(* Logix 5000 project; controller L3 vendor 1 type 14 code 92 rev 20.12; software revision 20.04; part 3 of 9 *)
(* tags used below, declared in another part *)
   B3 : DINT[100];
   N20 : DINT[200];
   N21 : DINT[200];
   N7 : DINT[200];
   N9 : DINT[200];   // niveau decapage vers lancy (n9[10) ;;N9[70]
   S_SP_DEC : DINT;
   T4 : TIMER[180];
(* _2_GENERAL, continued *)

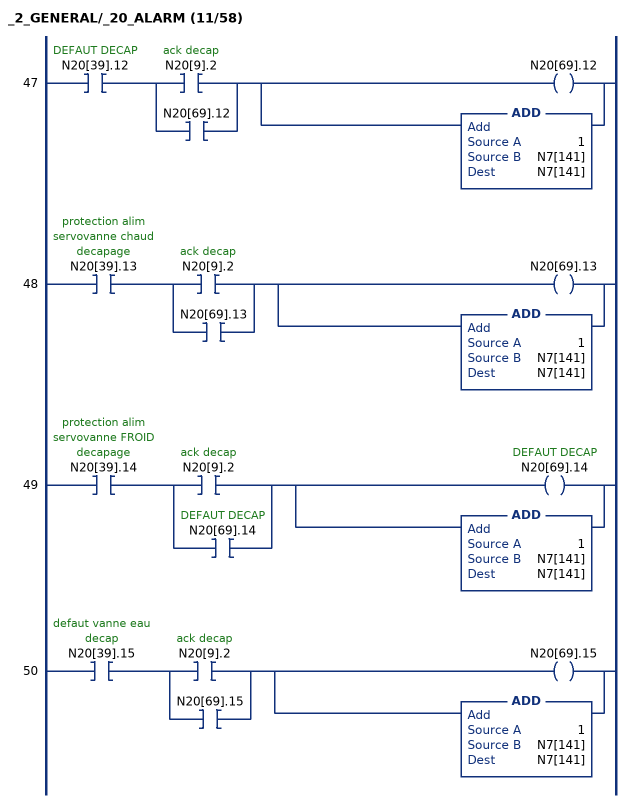
   [picture p26: _2_GENERAL/_20_ALARM rungs 47-50]
   47: XIC(N20[39].12)[XIC(N20[9].2) ,XIC(N20[69].12) ][OTE(N20[69].12) ,ADD(1,N7[141],N7[141]) ];
   48: XIC(N20[39].13)[XIC(N20[9].2) ,XIC(N20[69].13) ][OTE(N20[69].13) ,ADD(1,N7[141],N7[141]) ];
   49: XIC(N20[39].14)[XIC(N20[9].2) ,XIC(N20[69].14) ][OTE(N20[69].14) ,ADD(1,N7[141],N7[141]) ];
   50: XIC(N20[39].15)[XIC(N20[9].2) ,XIC(N20[69].15) ][OTE(N20[69].15) ,ADD(1,N7[141],N7[141]) ];
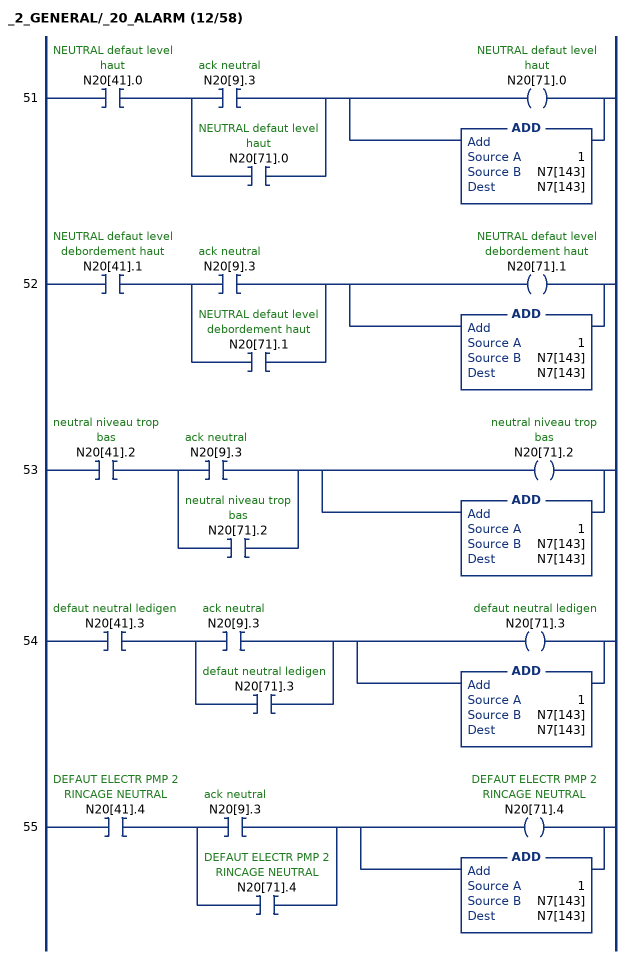
   51: XIC(N20[41].0)[XIC(N20[9].3) ,XIC(N20[71].0) ][OTE(N20[71].0) ,ADD(1,N7[143],N7[143]) ];
   52: XIC(N20[41].1)[XIC(N20[9].3) ,XIC(N20[71].1) ][OTE(N20[71].1) ,ADD(1,N7[143],N7[143]) ];
   53: XIC(N20[41].2)[XIC(N20[9].3) ,XIC(N20[71].2) ][OTE(N20[71].2) ,ADD(1,N7[143],N7[143]) ];
   54: XIC(N20[41].3)[XIC(N20[9].3) ,XIC(N20[71].3) ][OTE(N20[71].3) ,ADD(1,N7[143],N7[143]) ];
   55: XIC(N20[41].4)[XIC(N20[9].3) ,XIC(N20[71].4) ][OTE(N20[71].4) ,ADD(1,N7[143],N7[143]) ];
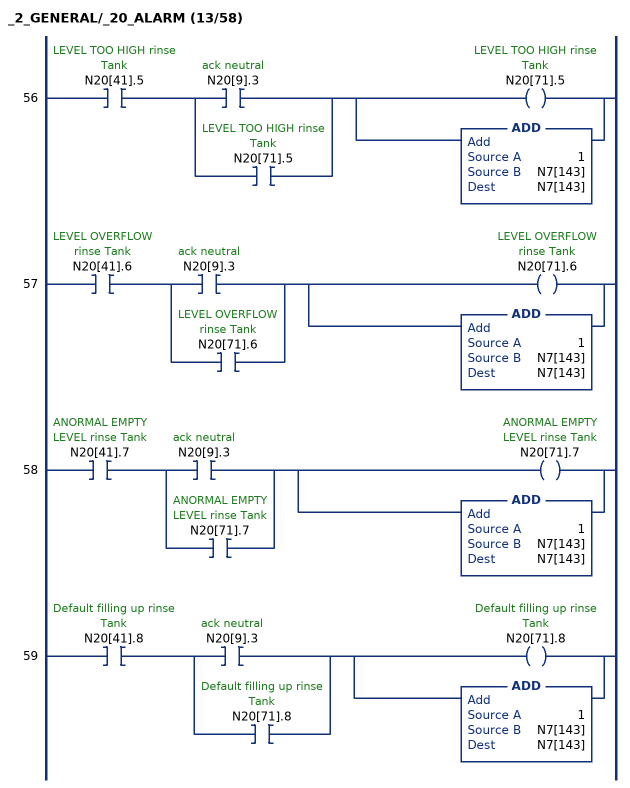
   56: XIC(N20[41].5)[XIC(N20[9].3) ,XIC(N20[71].5) ][OTE(N20[71].5) ,ADD(1,N7[143],N7[143]) ];
   57: XIC(N20[41].6)[XIC(N20[9].3) ,XIC(N20[71].6) ][OTE(N20[71].6) ,ADD(1,N7[143],N7[143]) ];
   58: XIC(N20[41].7)[XIC(N20[9].3) ,XIC(N20[71].7) ][OTE(N20[71].7) ,ADD(1,N7[143],N7[143]) ];
   59: XIC(N20[41].8)[XIC(N20[9].3) ,XIC(N20[71].8) ][OTE(N20[71].8) ,ADD(1,N7[143],N7[143]) ];
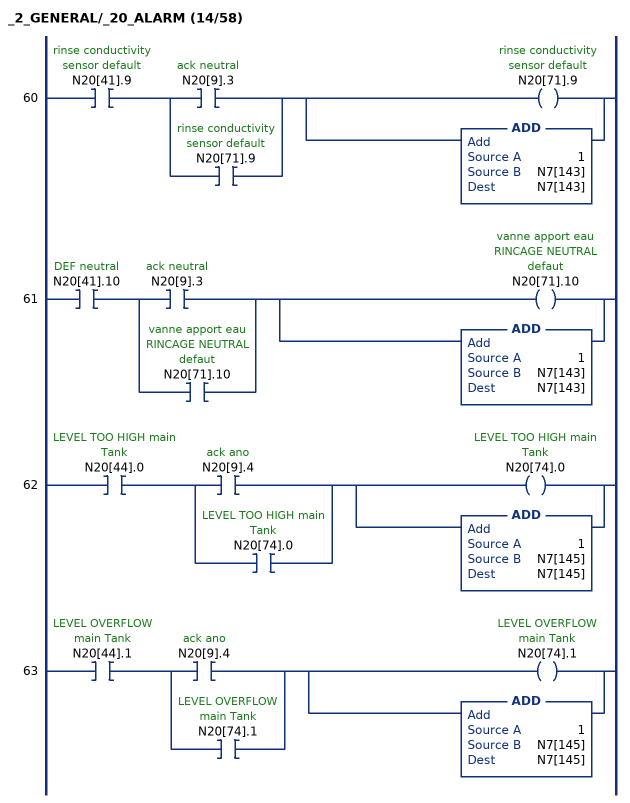
   60: XIC(N20[41].9)[XIC(N20[9].3) ,XIC(N20[71].9) ][OTE(N20[71].9) ,ADD(1,N7[143],N7[143]) ];
   61: XIC(N20[41].10)[XIC(N20[9].3) ,XIC(N20[71].10) ][OTE(N20[71].10) ,ADD(1,N7[143],N7[143]) ];
   62: XIC(N20[44].0)[XIC(N20[9].4) ,XIC(N20[74].0) ][OTE(N20[74].0) ,ADD(1,N7[145],N7[145]) ];
   63: XIC(N20[44].1)[XIC(N20[9].4) ,XIC(N20[74].1) ][OTE(N20[74].1) ,ADD(1,N7[145],N7[145]) ];
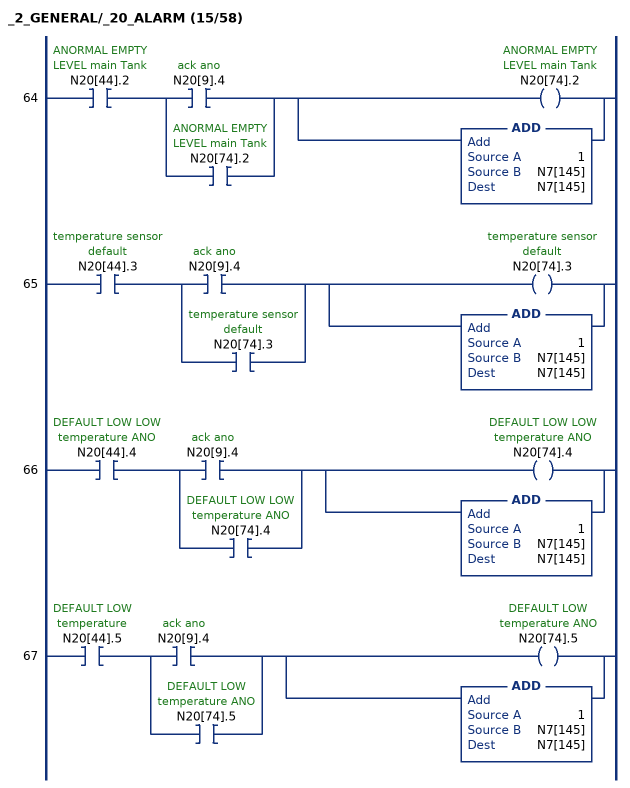
   64: XIC(N20[44].2)[XIC(N20[9].4) ,XIC(N20[74].2) ][OTE(N20[74].2) ,ADD(1,N7[145],N7[145]) ];
   65: XIC(N20[44].3)[XIC(N20[9].4) ,XIC(N20[74].3) ][OTE(N20[74].3) ,ADD(1,N7[145],N7[145]) ];
   66: XIC(N20[44].4)[XIC(N20[9].4) ,XIC(N20[74].4) ][OTE(N20[74].4) ,ADD(1,N7[145],N7[145]) ];
   67: XIC(N20[44].5)[XIC(N20[9].4) ,XIC(N20[74].5) ][OTE(N20[74].5) ,ADD(1,N7[145],N7[145]) ];
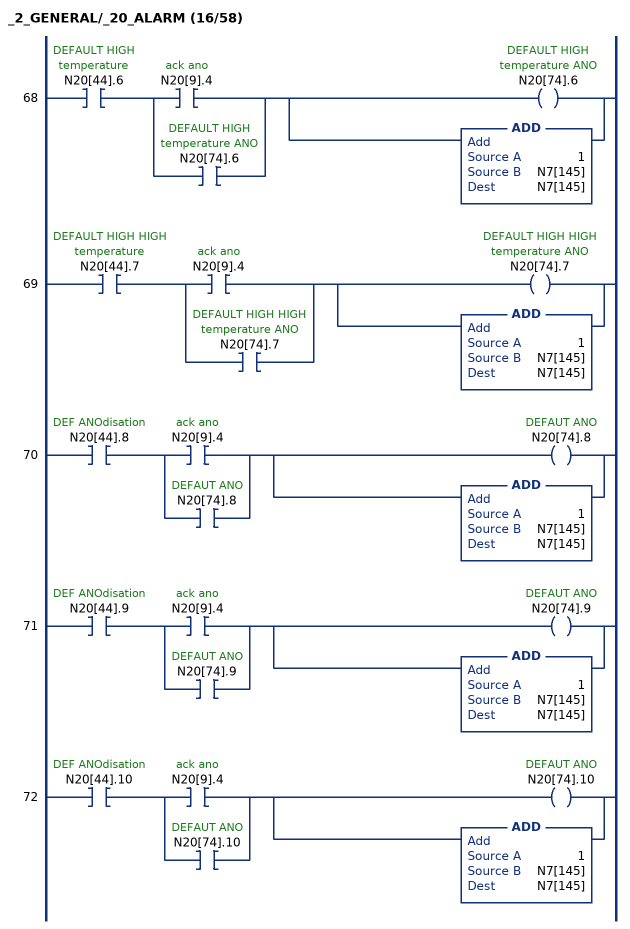
   68: XIC(N20[44].6)[XIC(N20[9].4) ,XIC(N20[74].6) ][OTE(N20[74].6) ,ADD(1,N7[145],N7[145]) ];
   69: XIC(N20[44].7)[XIC(N20[9].4) ,XIC(N20[74].7) ][OTE(N20[74].7) ,ADD(1,N7[145],N7[145]) ];
   70: XIC(N20[44].8)[XIC(N20[9].4) ,XIC(N20[74].8) ][OTE(N20[74].8) ,ADD(1,N7[145],N7[145]) ];
   71: XIC(N20[44].9)[XIC(N20[9].4) ,XIC(N20[74].9) ][OTE(N20[74].9) ,ADD(1,N7[145],N7[145]) ];
   72: XIC(N20[44].10)[XIC(N20[9].4) ,XIC(N20[74].10) ][OTE(N20[74].10) ,ADD(1,N7[145],N7[145]) ];
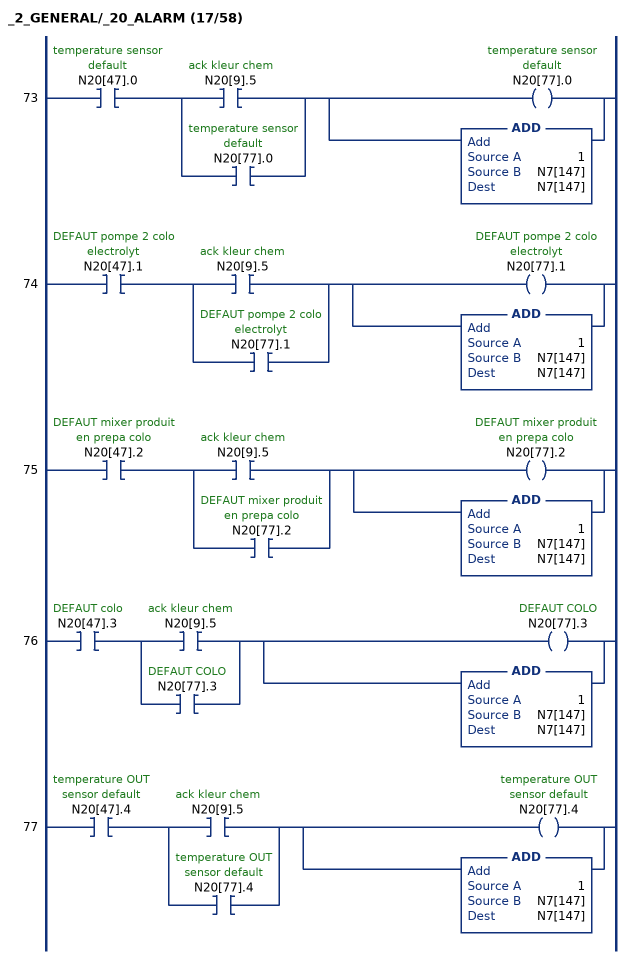
   73: XIC(N20[47].0)[XIC(N20[9].5) ,XIC(N20[77].0) ][OTE(N20[77].0) ,ADD(1,N7[147],N7[147]) ];
   74: XIC(N20[47].1)[XIC(N20[9].5) ,XIC(N20[77].1) ][OTE(N20[77].1) ,ADD(1,N7[147],N7[147]) ];
   75: XIC(N20[47].2)[XIC(N20[9].5) ,XIC(N20[77].2) ][OTE(N20[77].2) ,ADD(1,N7[147],N7[147]) ];
   76: XIC(N20[47].3)[XIC(N20[9].5) ,XIC(N20[77].3) ][OTE(N20[77].3) ,ADD(1,N7[147],N7[147]) ];
   77: XIC(N20[47].4)[XIC(N20[9].5) ,XIC(N20[77].4) ][OTE(N20[77].4) ,ADD(1,N7[147],N7[147]) ];
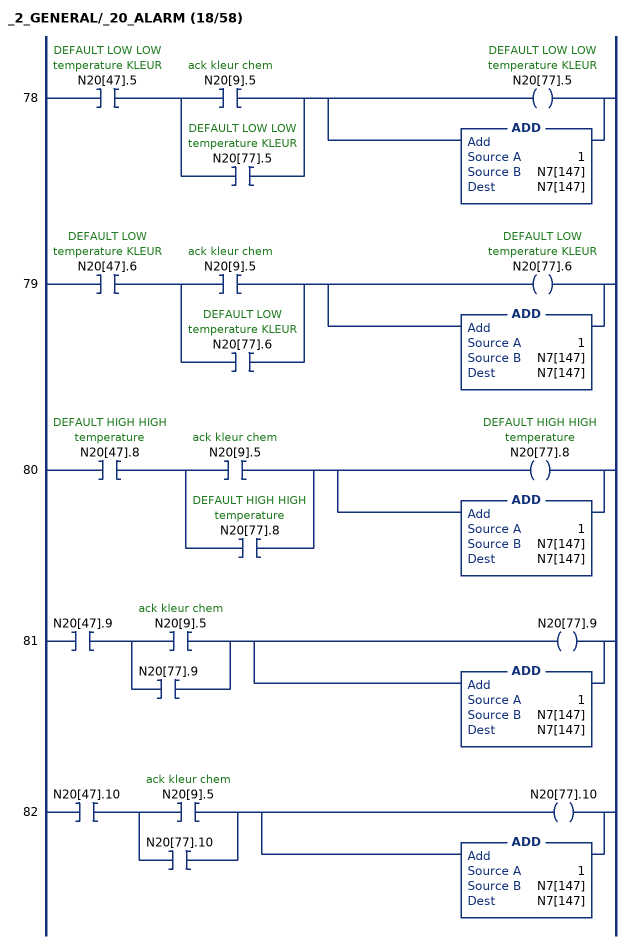
   78: XIC(N20[47].5)[XIC(N20[9].5) ,XIC(N20[77].5) ][OTE(N20[77].5) ,ADD(1,N7[147],N7[147]) ];
   79: XIC(N20[47].6)[XIC(N20[9].5) ,XIC(N20[77].6) ][OTE(N20[77].6) ,ADD(1,N7[147],N7[147]) ];
   80: XIC(N20[47].8)[XIC(N20[9].5) ,XIC(N20[77].8) ][OTE(N20[77].8) ,ADD(1,N7[147],N7[147]) ];
   81: XIC(N20[47].9)[XIC(N20[9].5) ,XIC(N20[77].9) ][OTE(N20[77].9) ,ADD(1,N7[147],N7[147]) ];
   82: XIC(N20[47].10)[XIC(N20[9].5) ,XIC(N20[77].10) ][OTE(N20[77].10) ,ADD(1,N7[147],N7[147]) ];
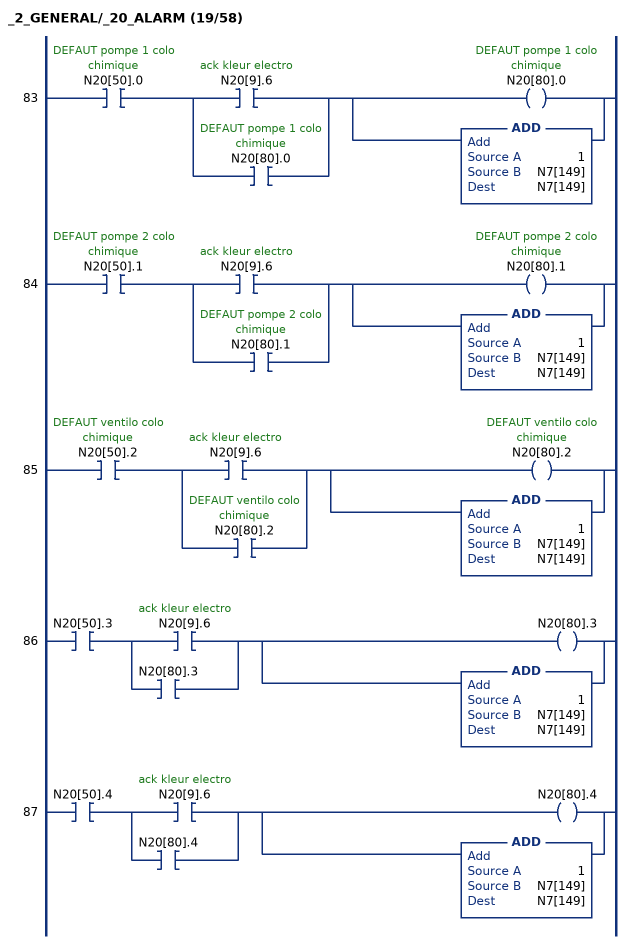
   83: XIC(N20[50].0)[XIC(N20[9].6) ,XIC(N20[80].0) ][OTE(N20[80].0) ,ADD(1,N7[149],N7[149]) ];
   84: XIC(N20[50].1)[XIC(N20[9].6) ,XIC(N20[80].1) ][OTE(N20[80].1) ,ADD(1,N7[149],N7[149]) ];
   85: XIC(N20[50].2)[XIC(N20[9].6) ,XIC(N20[80].2) ][OTE(N20[80].2) ,ADD(1,N7[149],N7[149]) ];
   86: XIC(N20[50].3)[XIC(N20[9].6) ,XIC(N20[80].3) ][OTE(N20[80].3) ,ADD(1,N7[149],N7[149]) ];
   87: XIC(N20[50].4)[XIC(N20[9].6) ,XIC(N20[80].4) ][OTE(N20[80].4) ,ADD(1,N7[149],N7[149]) ];
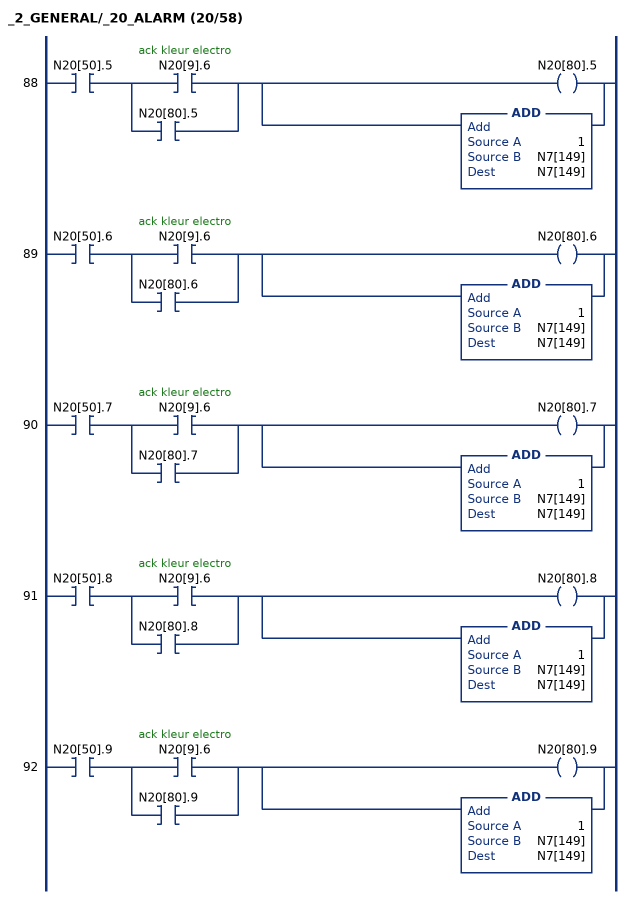
   88: XIC(N20[50].5)[XIC(N20[9].6) ,XIC(N20[80].5) ][OTE(N20[80].5) ,ADD(1,N7[149],N7[149]) ];
   89: XIC(N20[50].6)[XIC(N20[9].6) ,XIC(N20[80].6) ][OTE(N20[80].6) ,ADD(1,N7[149],N7[149]) ];
   90: XIC(N20[50].7)[XIC(N20[9].6) ,XIC(N20[80].7) ][OTE(N20[80].7) ,ADD(1,N7[149],N7[149]) ];
   91: XIC(N20[50].8)[XIC(N20[9].6) ,XIC(N20[80].8) ][OTE(N20[80].8) ,ADD(1,N7[149],N7[149]) ];
   92: XIC(N20[50].9)[XIC(N20[9].6) ,XIC(N20[80].9) ][OTE(N20[80].9) ,ADD(1,N7[149],N7[149]) ];
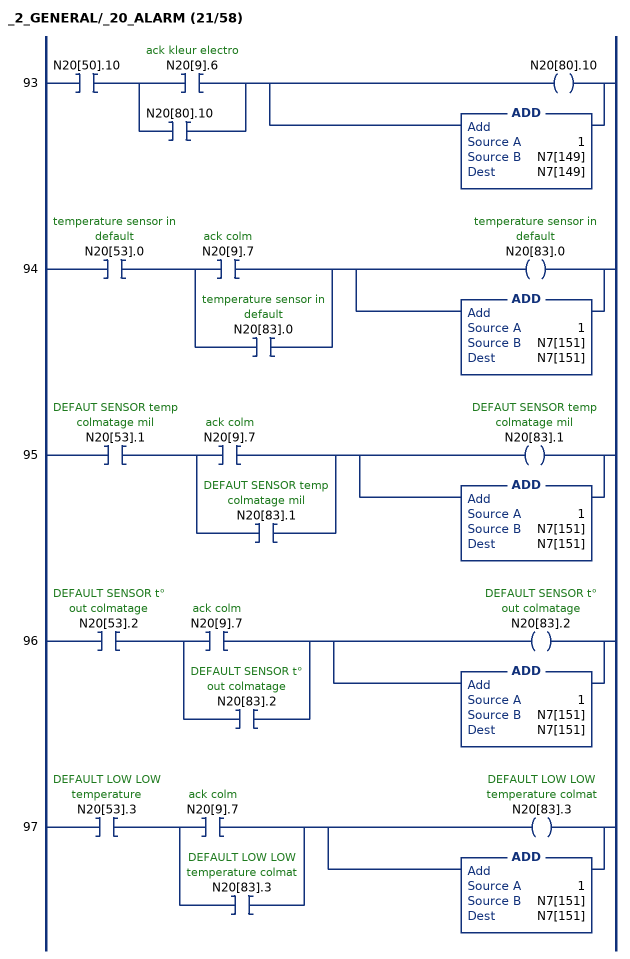
   93: XIC(N20[50].10)[XIC(N20[9].6) ,XIC(N20[80].10) ][OTE(N20[80].10) ,ADD(1,N7[149],N7[149]) ];
   94: XIC(N20[53].0)[XIC(N20[9].7) ,XIC(N20[83].0) ][OTE(N20[83].0) ,ADD(1,N7[151],N7[151]) ];
   95: XIC(N20[53].1)[XIC(N20[9].7) ,XIC(N20[83].1) ][OTE(N20[83].1) ,ADD(1,N7[151],N7[151]) ];
   96: XIC(N20[53].2)[XIC(N20[9].7) ,XIC(N20[83].2) ][OTE(N20[83].2) ,ADD(1,N7[151],N7[151]) ];
   97: XIC(N20[53].3)[XIC(N20[9].7) ,XIC(N20[83].3) ][OTE(N20[83].3) ,ADD(1,N7[151],N7[151]) ];
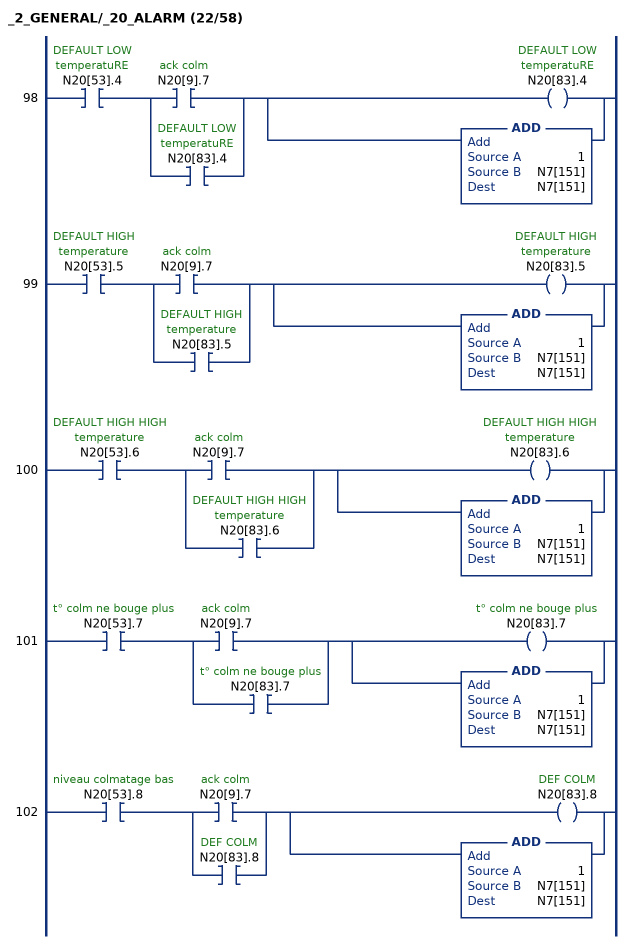
   98: XIC(N20[53].4)[XIC(N20[9].7) ,XIC(N20[83].4) ][OTE(N20[83].4) ,ADD(1,N7[151],N7[151]) ];
   99: XIC(N20[53].5)[XIC(N20[9].7) ,XIC(N20[83].5) ][OTE(N20[83].5) ,ADD(1,N7[151],N7[151]) ];
   100: XIC(N20[53].6)[XIC(N20[9].7) ,XIC(N20[83].6) ][OTE(N20[83].6) ,ADD(1,N7[151],N7[151]) ];
   101: XIC(N20[53].7)[XIC(N20[9].7) ,XIC(N20[83].7) ][OTE(N20[83].7) ,ADD(1,N7[151],N7[151]) ];
   102: XIC(N20[53].8)[XIC(N20[9].7) ,XIC(N20[83].8) ][OTE(N20[83].8) ,ADD(1,N7[151],N7[151]) ];
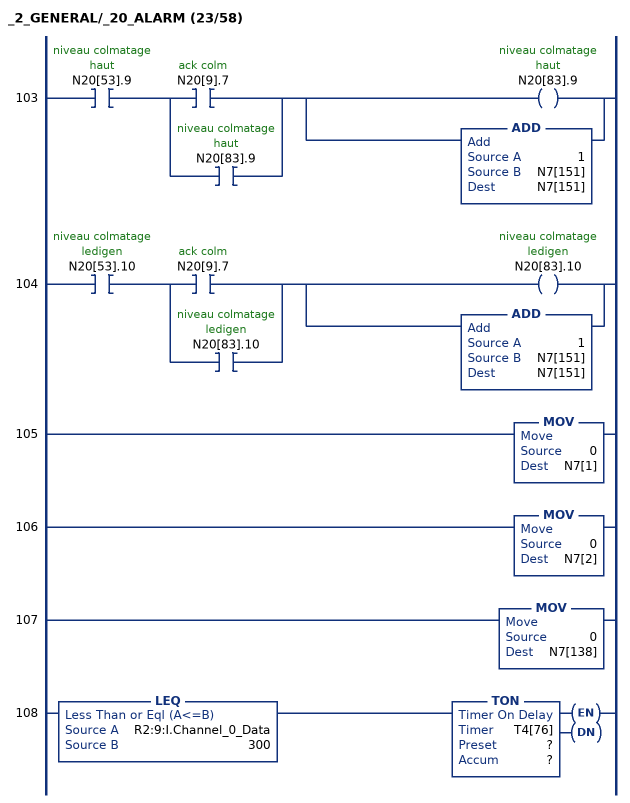
   103: XIC(N20[53].9)[XIC(N20[9].7) ,XIC(N20[83].9) ][OTE(N20[83].9) ,ADD(1,N7[151],N7[151]) ];
   104: XIC(N20[53].10)[XIC(N20[9].7) ,XIC(N20[83].10) ][OTE(N20[83].10) ,ADD(1,N7[151],N7[151]) ];
   105: MOV(0,N7[1]);
   106: MOV(0,N7[2]);
   107: MOV(0,N7[138]);
   108: LEQ(R2:9:I.Channel_0_Data,300)TON(T4[76],?,?);
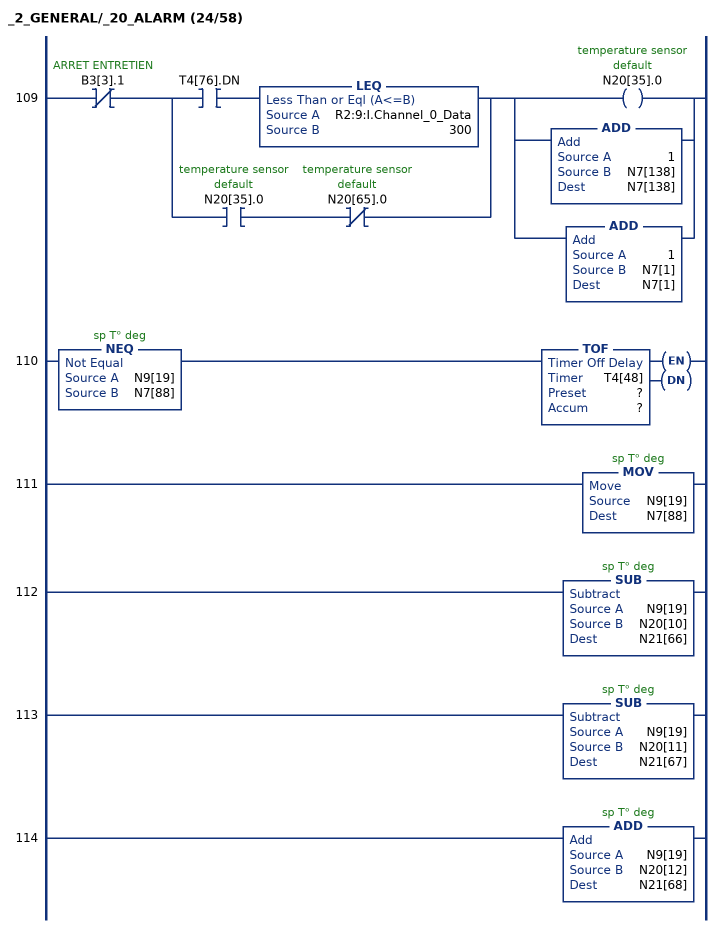
   109: XIO(B3[3].1)[XIC(T4[76].DN) LEQ(R2:9:I.Channel_0_Data,300) ,XIC(N20[35].0) XIO(N20[65].0) ][OTE(N20[35].0) ,ADD(1,N7[138],N7[138]) ,ADD(1,N7[1],N7[1]) ];
   110: NEQ(N9[19],N7[88])TOF(T4[48],?,?);
   111: MOV(N9[19],N7[88]);
   112: SUB(N9[19],N20[10],N21[66]);
   113: SUB(N9[19],N20[11],N21[67]);
   114: ADD(N9[19],N20[12],N21[68]);
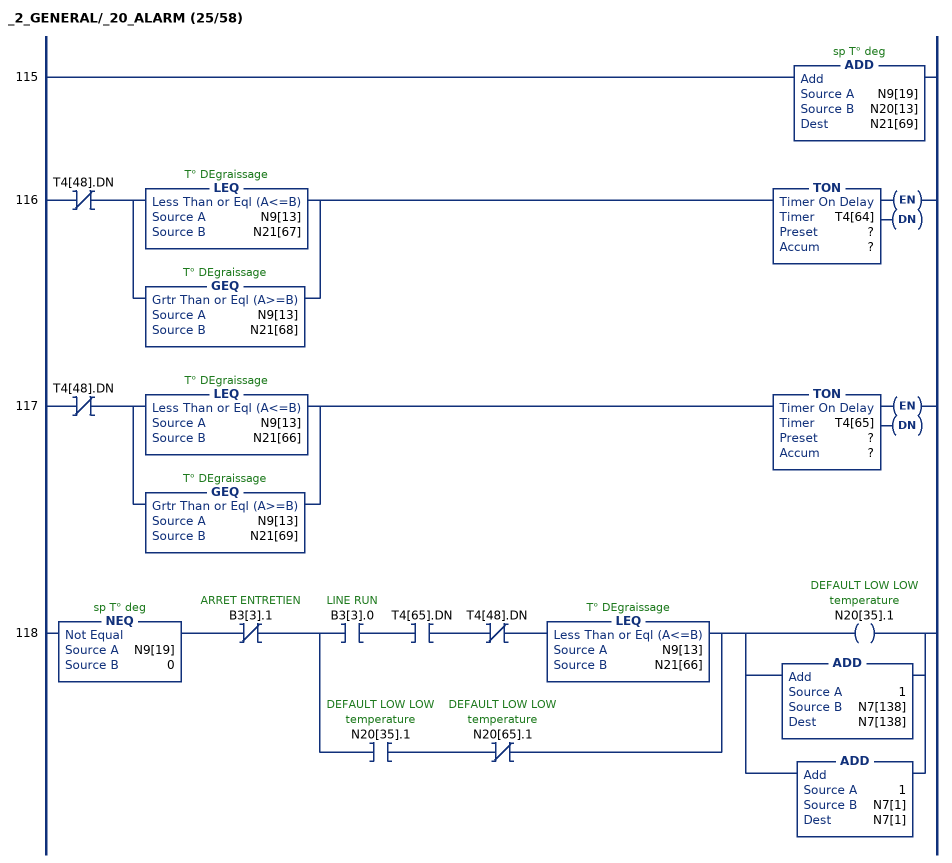
   115: ADD(N9[19],N20[13],N21[69]);
   116: XIO(T4[48].DN)[LEQ(N9[13],N21[67]) ,GEQ(N9[13],N21[68]) ]TON(T4[64],?,?);
   117: XIO(T4[48].DN)[LEQ(N9[13],N21[66]) ,GEQ(N9[13],N21[69]) ]TON(T4[65],?,?);
   118: NEQ(N9[19],0)XIO(B3[3].1)[XIC(B3[3].0) XIC(T4[65].DN) XIO(T4[48].DN) LEQ(N9[13],N21[66]) ,XIC(N20[35].1) XIO(N20[65].1) ][OTE(N20[35].1) ,ADD(1,N7[138],N7[138]) ,ADD(1,N7[1],N7[1]) ];
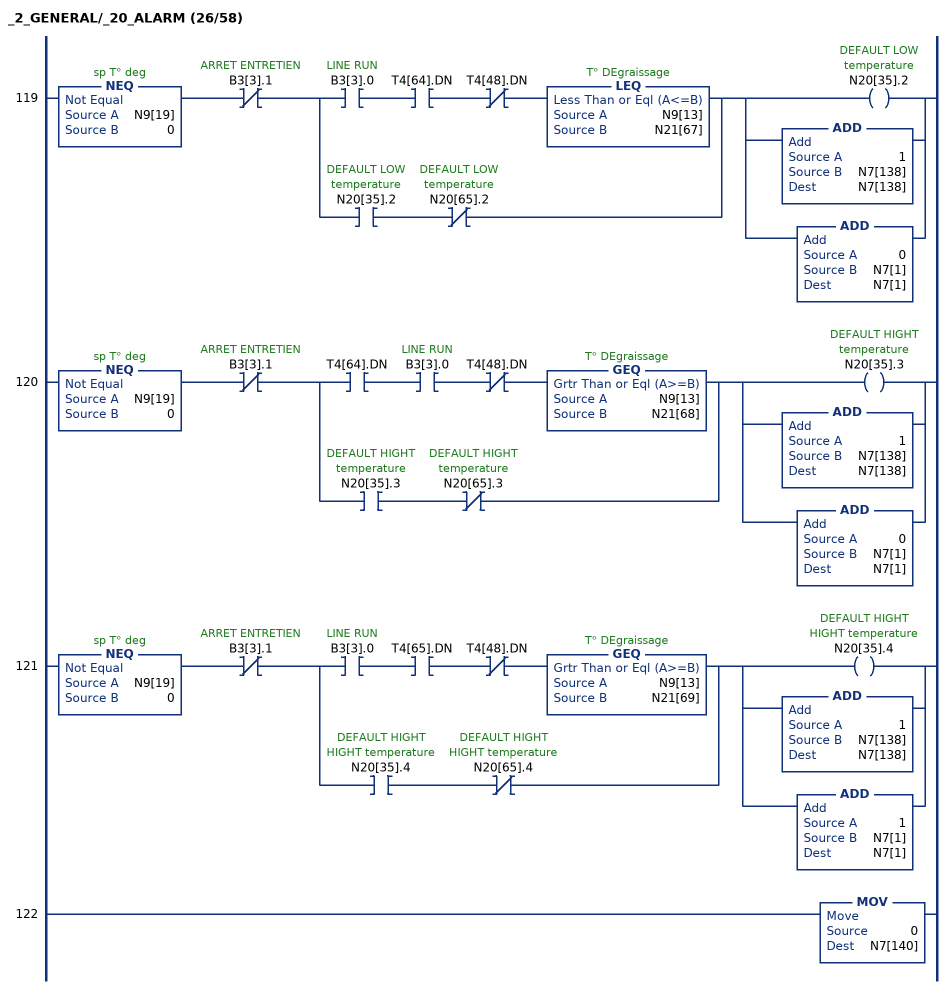
   119: NEQ(N9[19],0)XIO(B3[3].1)[XIC(B3[3].0) XIC(T4[64].DN) XIO(T4[48].DN) LEQ(N9[13],N21[67]) ,XIC(N20[35].2) XIO(N20[65].2) ][OTE(N20[35].2) ,ADD(1,N7[138],N7[138]) ,ADD(0,N7[1],N7[1]) ];
   120: NEQ(N9[19],0)XIO(B3[3].1)[XIC(T4[64].DN) XIC(B3[3].0) XIO(T4[48].DN) GEQ(N9[13],N21[68]) ,XIC(N20[35].3) XIO(N20[65].3) ][OTE(N20[35].3) ,ADD(1,N7[138],N7[138]) ,ADD(0,N7[1],N7[1]) ];
   121: NEQ(N9[19],0)XIO(B3[3].1)[XIC(B3[3].0) XIC(T4[65].DN) XIO(T4[48].DN) GEQ(N9[13],N21[69]) ,XIC(N20[35].4) XIO(N20[65].4) ][OTE(N20[35].4) ,ADD(1,N7[138],N7[138]) ,ADD(1,N7[1],N7[1]) ];
   122: MOV(0,N7[140]);
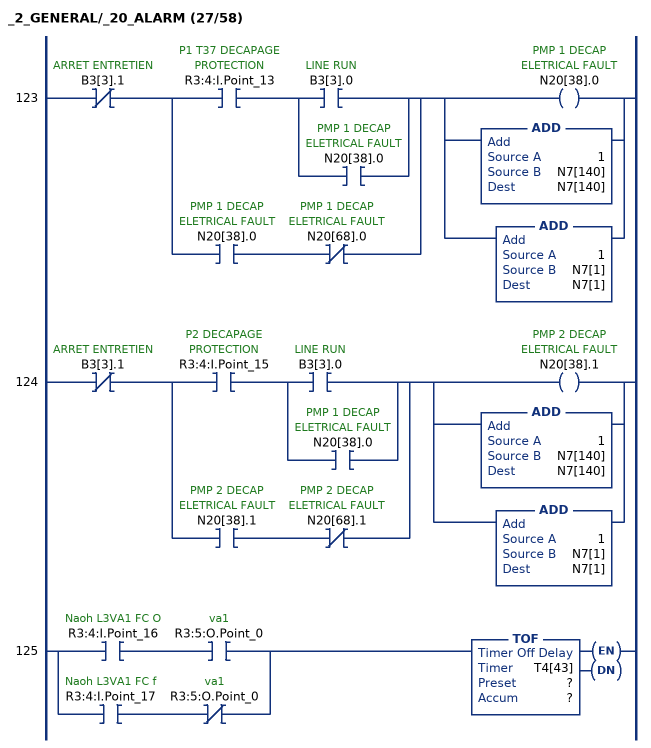
   123: XIO(B3[3].1)[XIC(R3:4:I.Point_13) [XIC(B3[3].0) ,XIC(N20[38].0) ] ,XIC(N20[38].0) XIO(N20[68].0) ][OTE(N20[38].0) ,ADD(1,N7[140],N7[140]) ,ADD(1,N7[1],N7[1]) ];
   124: XIO(B3[3].1)[XIC(R3:4:I.Point_15) [XIC(B3[3].0) ,XIC(N20[38].0) ] ,XIC(N20[38].1) XIO(N20[68].1) ][OTE(N20[38].1) ,ADD(1,N7[140],N7[140]) ,ADD(1,N7[1],N7[1]) ];
   125: [XIC(R3:4:I.Point_16) XIC(R3:5:O.Point_0) ,XIC(R3:4:I.Point_17) XIO(R3:5:O.Point_0) ]TOF(T4[43],?,?);
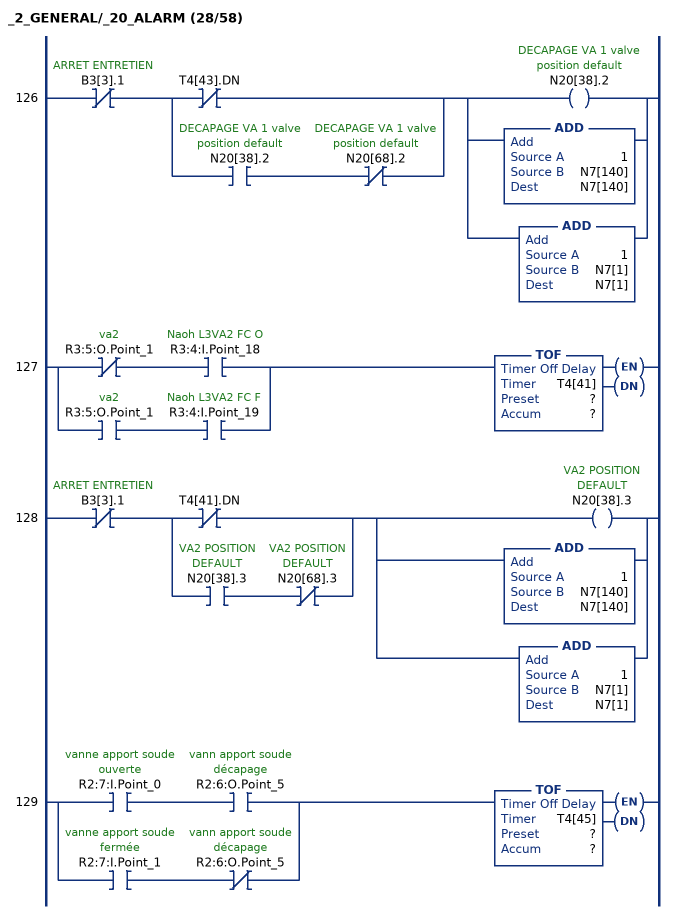
   126: XIO(B3[3].1)[XIO(T4[43].DN) ,XIC(N20[38].2) XIO(N20[68].2) ][OTE(N20[38].2) ,ADD(1,N7[140],N7[140]) ,ADD(1,N7[1],N7[1]) ];
   127: [XIO(R3:5:O.Point_1) XIC(R3:4:I.Point_18) ,XIC(R3:5:O.Point_1) XIC(R3:4:I.Point_19) ]TOF(T4[41],?,?);
   128: XIO(B3[3].1)[XIO(T4[41].DN) ,XIC(N20[38].3) XIO(N20[68].3) ][OTE(N20[38].3) ,ADD(1,N7[140],N7[140]) ,ADD(1,N7[1],N7[1]) ];
   129: [XIC(R2:7:I.Point_0) XIC(R2:6:O.Point_5) ,XIC(R2:7:I.Point_1) XIO(R2:6:O.Point_5) ]TOF(T4[45],?,?);
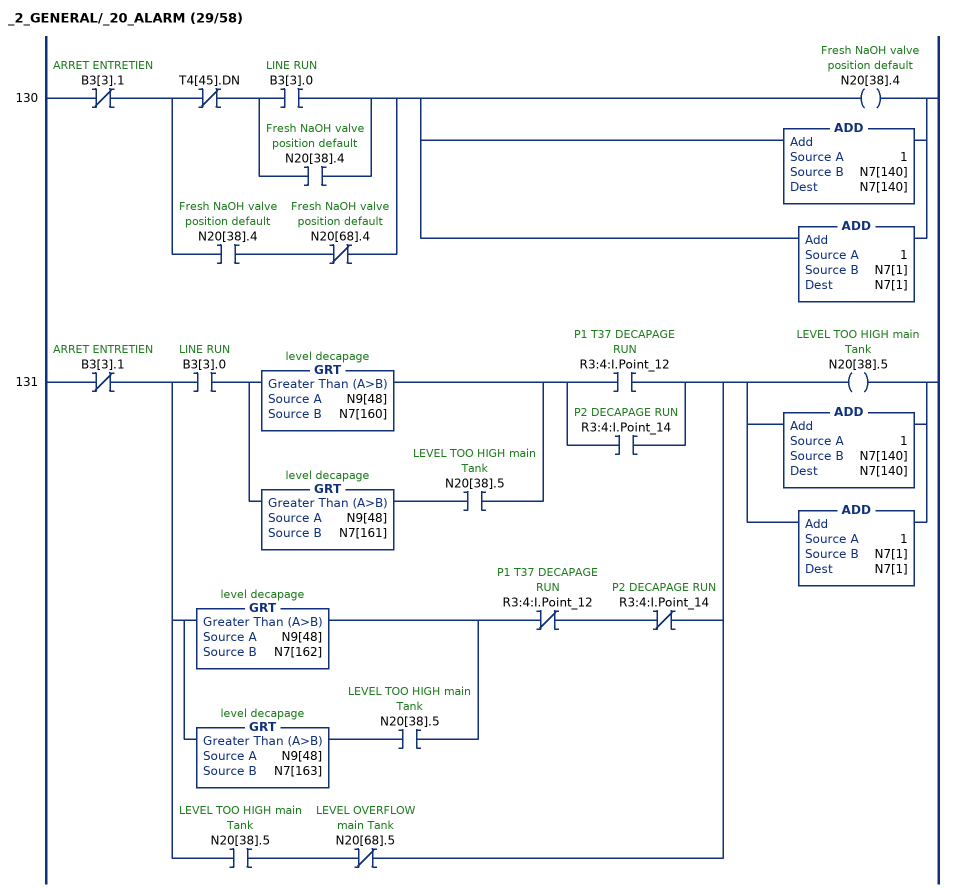
   130: XIO(B3[3].1)[XIO(T4[45].DN) [XIC(B3[3].0) ,XIC(N20[38].4) ] ,XIC(N20[38].4) XIO(N20[68].4) ][OTE(N20[38].4) ,ADD(1,N7[140],N7[140]) ,ADD(1,N7[1],N7[1]) ];
   131: XIO(B3[3].1)[XIC(B3[3].0) [GRT(N9[48],N7[160]) ,GRT(N9[48],N7[161]) XIC(N20[38].5) ] [XIC(R3:4:I.Point_12) ,XIC(R3:4:I.Point_14) ] ,[GRT(N9[48],N7[162]) ,GRT(N9[48],N7[163]) XIC(N20[38].5) ] XIO(R3:4:I.Point_12) XIO(R3:4:I.Point_14) ,XIC(N20[38].5) XIO(N20[68].5) ][OTE(N20[38].5) ,ADD(1,N7[140],N7[140]) ,ADD(1,N7[1],N7[1]) ];
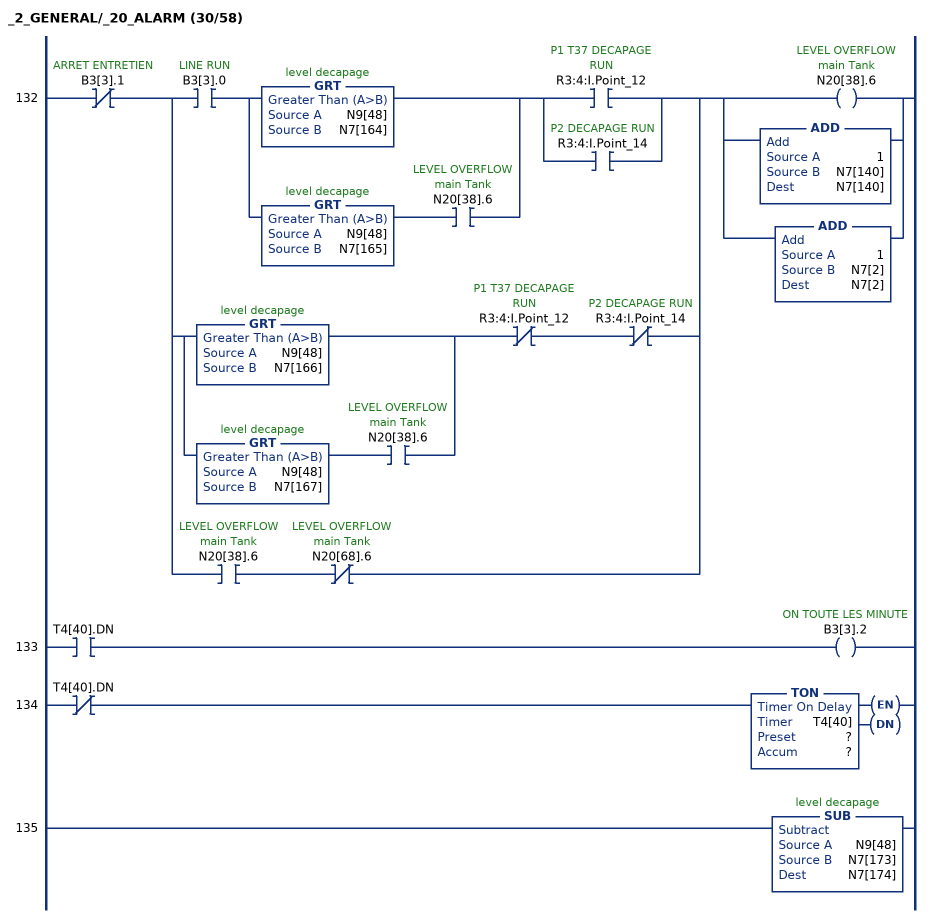
   132: XIO(B3[3].1)[XIC(B3[3].0) [GRT(N9[48],N7[164]) ,GRT(N9[48],N7[165]) XIC(N20[38].6) ] [XIC(R3:4:I.Point_12) ,XIC(R3:4:I.Point_14) ] ,[GRT(N9[48],N7[166]) ,GRT(N9[48],N7[167]) XIC(N20[38].6) ] XIO(R3:4:I.Point_12) XIO(R3:4:I.Point_14) ,XIC(N20[38].6) XIO(N20[68].6) ][OTE(N20[38].6) ,ADD(1,N7[140],N7[140]) ,ADD(1,N7[2],N7[2]) ];
   133: XIC(T4[40].DN)OTE(B3[3].2);
   134: XIO(T4[40].DN)TON(T4[40],?,?);
   135: SUB(N9[48],N7[173],N7[174]);
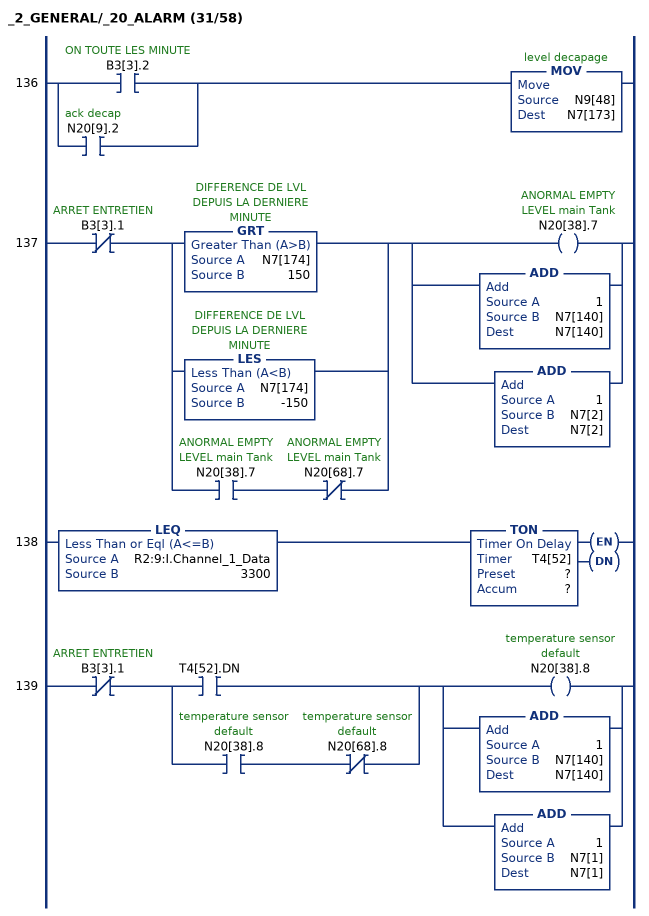
   136: [XIC(B3[3].2) ,XIC(N20[9].2) ]MOV(N9[48],N7[173]);
   137: XIO(B3[3].1)[GRT(N7[174],150) ,LES(N7[174],-150) ,XIC(N20[38].7) XIO(N20[68].7) ][OTE(N20[38].7) ,ADD(1,N7[140],N7[140]) ,ADD(1,N7[2],N7[2]) ];
   138: LEQ(R2:9:I.Channel_1_Data,3300)TON(T4[52],?,?);
   139: XIO(B3[3].1)[XIC(T4[52].DN) ,XIC(N20[38].8) XIO(N20[68].8) ][OTE(N20[38].8) ,ADD(1,N7[140],N7[140]) ,ADD(1,N7[1],N7[1]) ];
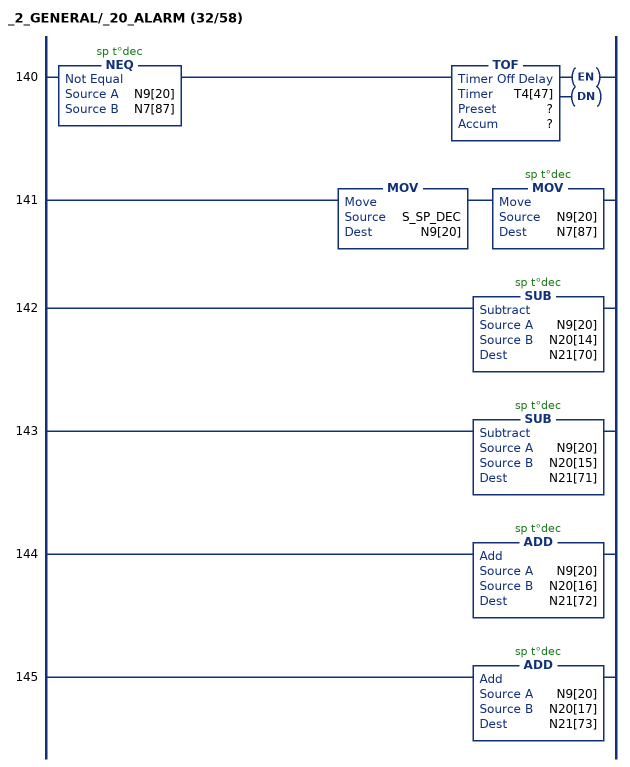
   140: NEQ(N9[20],N7[87])TOF(T4[47],?,?);
   141: MOV(S_SP_DEC,N9[20])MOV(N9[20],N7[87]);
   142: SUB(N9[20],N20[14],N21[70]);
   143: SUB(N9[20],N20[15],N21[71]);
   144: ADD(N9[20],N20[16],N21[72]);
   145: ADD(N9[20],N20[17],N21[73]);
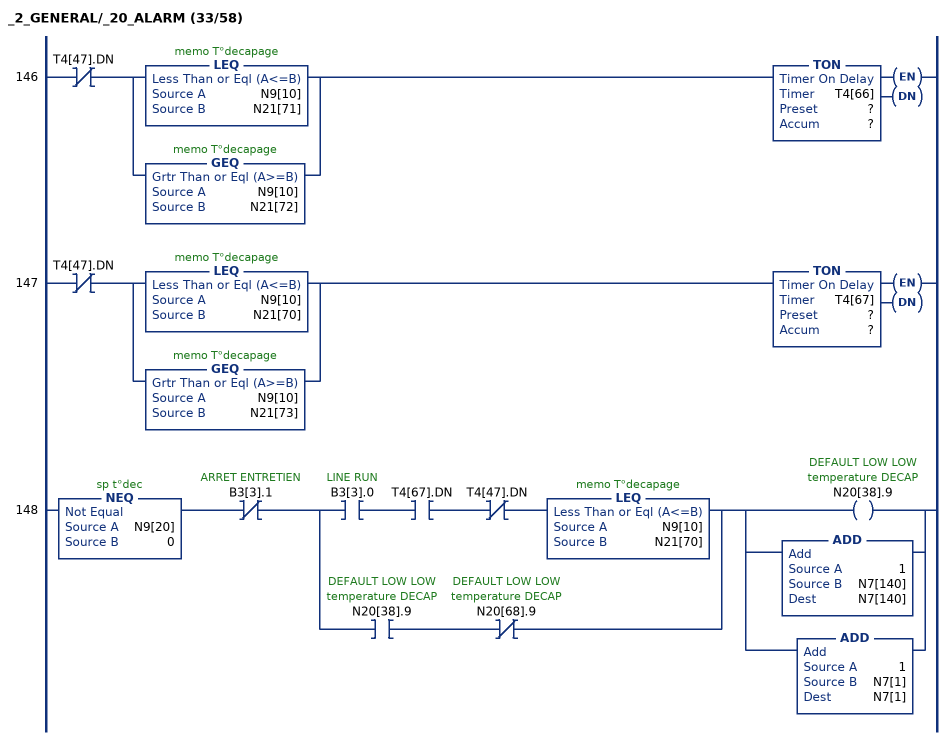
   146: XIO(T4[47].DN)[LEQ(N9[10],N21[71]) ,GEQ(N9[10],N21[72]) ]TON(T4[66],?,?);
   147: XIO(T4[47].DN)[LEQ(N9[10],N21[70]) ,GEQ(N9[10],N21[73]) ]TON(T4[67],?,?);
   148: NEQ(N9[20],0)XIO(B3[3].1)[XIC(B3[3].0) XIC(T4[67].DN) XIO(T4[47].DN) LEQ(N9[10],N21[70]) ,XIC(N20[38].9) XIO(N20[68].9) ][OTE(N20[38].9) ,ADD(1,N7[140],N7[140]) ,ADD(1,N7[1],N7[1]) ];
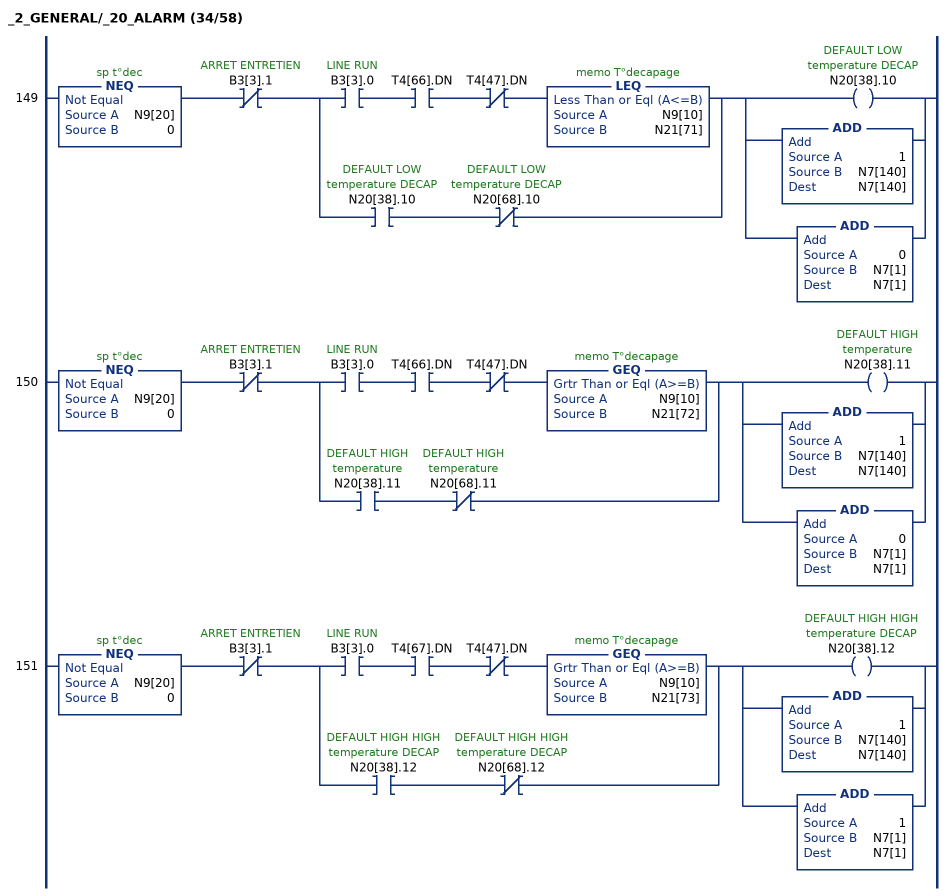
   149: NEQ(N9[20],0)XIO(B3[3].1)[XIC(B3[3].0) XIC(T4[66].DN) XIO(T4[47].DN) LEQ(N9[10],N21[71]) ,XIC(N20[38].10) XIO(N20[68].10) ][OTE(N20[38].10) ,ADD(1,N7[140],N7[140]) ,ADD(0,N7[1],N7[1]) ];
   150: NEQ(N9[20],0)XIO(B3[3].1)[XIC(B3[3].0) XIC(T4[66].DN) XIO(T4[47].DN) GEQ(N9[10],N21[72]) ,XIC(N20[38].11) XIO(N20[68].11) ][OTE(N20[38].11) ,ADD(1,N7[140],N7[140]) ,ADD(0,N7[1],N7[1]) ];
   151: NEQ(N9[20],0)XIO(B3[3].1)[XIC(B3[3].0) XIC(T4[67].DN) XIO(T4[47].DN) GEQ(N9[10],N21[73]) ,XIC(N20[38].12) XIO(N20[68].12) ][OTE(N20[38].12) ,ADD(1,N7[140],N7[140]) ,ADD(1,N7[1],N7[1]) ];
